// TIA Portal V17 export
// export: Created 2022-07-20T06:59:51.3246087Z, ExportSetting WithDefaults, DisplayName Totally Integrated Automation Portal, DisplayVersion V17, DisplayName TIA Portal Openness, DisplayVersion V17, DisplayName TIA Portal Version Control Interface, DisplayVersion V17, DisplayName SINAMICS Startdrive Advanced, DisplayVersion V17, DisplayName SINAMICS Startdrive G130, G150, S120, S150, SINAMICS MV, S210, DisplayVersion V17, DisplayName SINAMICS Startdrive G110M, G120, G120C, G120D, G120P, G115D, DisplayVersion V17, DisplayName STEP 7 Professional, DisplayVersion V17, DisplayName STEP 7 Safety, DisplayVersion V17, DisplayName WinCC Advanced, DisplayVersion V17
FUNCTION_BLOCK "FB10066_IperAirSystem"   // FB10066, LAD
{ S7_Optimized_Access := 'TRUE' }
VERSION : 0.1
// stored: AutoNumber false, IsIECCheckEnabled false, IsRetainMemResEnabled false, MemoryReserve 100, SetENOAutomatically false, UDAEnableTagReadback false
   VAR_INPUT
      Acknwoledge : Bool;
      TankOverPressureTime : Time;
      EmptyClusterOverPressureTime : Time;
      RequestTankOverpressure : Bool;
      RequestEmptyClusterOverpressure : Bool;
      RequestEmptyClusterOverpressure_1 : Bool;
      RequestEmptyClusterOverpressure_2 : Bool;
      RequestEmptyClusterOverpressure_3 : Bool;
      RequestEmptyClusterOverpressure_4 : Bool;
      RequestEmptyClusterOverpressure_5 : Bool;
      RequestEmptyClusterOverpressure_6 : Bool;
   END_VAR
   VAR_OUTPUT
      ActiveTankPurgeSolenoideValve : Bool;
      ActiveEmptyClusterPurgeSolenoidValve_1 : Bool;
      ActiveEmptyClusterPurgeSolenoidValve_2 : Bool;
      ActiveEmptyClusterPurgeSolenoidValve_3 : Bool;
      ActiveEmptyClusterPurgeSolenoidValve_4 : Bool;
      ActiveEmptyClusterPurgeSolenoidValve_5 : Bool;
      ActiveEmptyClusterPurgeSolenoidValve_6 : Bool;
      EmptyClusterOverpressureDone : Bool;
      TankOverpressureDone : Bool;
   END_VAR
   VAR
      ClusterInkCircuitStateDiagram : Int;
      R_TRIG_RequestTankOverpressure : R_TRIG;
      R_TRIG_RequestClusterOverpressure { S7_SetPoint := 'True'} : R_TRIG;
      F_TRIG_RequestTankOverpressure : F_TRIG;
      F_TRIG_RequestEmptyClusterOverpressure { S7_SetPoint := 'True'} : F_TRIG;
      TON_TankOverpressure { S7_SetPoint := 'True'} : TON_TIME;
      TON_EmptyClusterOverpressure { S7_SetPoint := 'True'} : TON_TIME;
   END_VAR
   VAR CONSTANT
      WAIT_FOR_CLUSTER_INK_CIRCUIT_REQUESTS : Int := 0;
      OVERPRESSURE_TANK : Int := 10;
      OVERPRESSURE_EMPTYCLUSTER : Int := 20;
      CLUSTER_INK_CIRCUIT_REQUESTS_DONE : Int := 30;
      "==========" : Bool;
   END_VAR
BEGIN

REGION Network 1 (SCL): First Scan
   IF "FirstScan" THEN
       #TankOverpressureDone := FALSE;
       #EmptyClusterOverpressureDone := FALSE;
   END_IF;
END_REGION

REGION Network 2 (SCL): Edge Signals & Timers
   REGION EDGE SIGNALS
       #R_TRIG_RequestTankOverpressure(CLK := #RequestTankOverpressure);
       #R_TRIG_RequestClusterOverpressure(CLK := #RequestEmptyClusterOverpressure);

       #F_TRIG_RequestTankOverpressure(CLK := #RequestTankOverpressure);
       #F_TRIG_RequestEmptyClusterOverpressure(CLK := #RequestEmptyClusterOverpressure);
   END_REGION

   REGION TIMERS
       #TON_TankOverpressure(IN := #ClusterInkCircuitStateDiagram = #OVERPRESSURE_TANK,
                             PT := #TankOverPressureTime);

       #TON_EmptyClusterOverpressure(IN := #ClusterInkCircuitStateDiagram = #OVERPRESSURE_EMPTYCLUSTER,
                                     PT := #EmptyClusterOverPressureTime);
   END_REGION
END_REGION

REGION Network 3 (SCL): Cluster Ink Circuit Management
   CASE #ClusterInkCircuitStateDiagram OF
       #WAIT_FOR_CLUSTER_INK_CIRCUIT_REQUESTS:  
           IF #R_TRIG_RequestTankOverpressure.Q THEN
               #TankOverpressureDone := FALSE;
               #ClusterInkCircuitStateDiagram := #OVERPRESSURE_TANK;
           ELSIF #R_TRIG_RequestClusterOverpressure.Q THEN
               #EmptyClusterOverpressureDone := FALSE;
               #ClusterInkCircuitStateDiagram := #OVERPRESSURE_EMPTYCLUSTER;
           END_IF;
       #OVERPRESSURE_TANK:  
           #ActiveTankPurgeSolenoideValve := TRUE;
           IF #TON_TankOverpressure.Q OR #F_TRIG_RequestTankOverpressure.Q THEN
               #ActiveTankPurgeSolenoideValve := FALSE;
               #TankOverpressureDone := TRUE;
               #ClusterInkCircuitStateDiagram := #CLUSTER_INK_CIRCUIT_REQUESTS_DONE;
           END_IF;
       #OVERPRESSURE_EMPTYCLUSTER:
           IF #RequestEmptyClusterOverpressure_1 THEN
               #ActiveEmptyClusterPurgeSolenoidValve_1 := TRUE;
           ELSE
               #ActiveEmptyClusterPurgeSolenoidValve_1 := FALSE;
           END_IF;

           IF #RequestEmptyClusterOverpressure_2 THEN
               #ActiveEmptyClusterPurgeSolenoidValve_2 := TRUE;
           ELSE
               #ActiveEmptyClusterPurgeSolenoidValve_2 := FALSE;
           END_IF;

           IF #RequestEmptyClusterOverpressure_3 THEN
               #ActiveEmptyClusterPurgeSolenoidValve_3 := TRUE;
           ELSE
               #ActiveEmptyClusterPurgeSolenoidValve_3 := FALSE;
           END_IF;

           IF #RequestEmptyClusterOverpressure_4 THEN
               #ActiveEmptyClusterPurgeSolenoidValve_4 := TRUE;
           ELSE
               #ActiveEmptyClusterPurgeSolenoidValve_4 := FALSE;
           END_IF;

           IF #RequestEmptyClusterOverpressure_5 THEN
               #ActiveEmptyClusterPurgeSolenoidValve_5 := TRUE;
           ELSE
               #ActiveEmptyClusterPurgeSolenoidValve_5 := FALSE;
           END_IF;

           IF #RequestEmptyClusterOverpressure_6 THEN
               #ActiveEmptyClusterPurgeSolenoidValve_6 := TRUE;
           ELSE
               #ActiveEmptyClusterPurgeSolenoidValve_6 := FALSE;
           END_IF;

           IF #TON_EmptyClusterOverpressure.Q OR #F_TRIG_RequestEmptyClusterOverpressure.Q THEN
               #ActiveEmptyClusterPurgeSolenoidValve_1 := FALSE;
               #ActiveEmptyClusterPurgeSolenoidValve_2 := FALSE;
               #ActiveEmptyClusterPurgeSolenoidValve_3 := FALSE;
               #ActiveEmptyClusterPurgeSolenoidValve_4 := FALSE;
               #ActiveEmptyClusterPurgeSolenoidValve_5 := FALSE;
               #ActiveEmptyClusterPurgeSolenoidValve_6 := FALSE;
               #EmptyClusterOverpressureDone := TRUE;
               #ClusterInkCircuitStateDiagram := #CLUSTER_INK_CIRCUIT_REQUESTS_DONE;
           END_IF;
       #CLUSTER_INK_CIRCUIT_REQUESTS_DONE:
           #ClusterInkCircuitStateDiagram := #WAIT_FOR_CLUSTER_INK_CIRCUIT_REQUESTS;
   END_CASE;
END_REGION
END_FUNCTION_BLOCK
